// Mitsubishi GX Works2 project: BookEX6_11 Trig   PLC: Q13UDV

// global labels: Global
VAR_GLOBAL
  bVar0 AT M5000 : BOOL;
  abArray0 AT M5010 : ARRAY [0..49] OF BOOL;
  sStr0 AT D5000 : STRING[199];
  sStr1 AT D5100 : STRING[199];
  sStr2 AT D5200 : STRING[199];
  sStr3 AT D5300 : STRING[199];
  sStr4 AT D5400 : STRING[199];
  sStr5 AT D5500 : STRING[199];
  sStr6 AT D5600 : STRING[199];
  sStr7 AT D5700 : STRING[199];
  sStr8 AT D5800 : STRING[199];
  sStr9 AT D5900 : STRING[199];
  iVar0 AT D4500 : INT;
  iVar1 AT D4501 : INT;
  iVar2 AT D4502 : INT;
  iVar3 AT D4503 : INT;
  iVar4 AT D4504 : INT;
  iVar5 AT D4505 : INT;
  iVar6 AT D4506 : INT;
  iVar7 AT D4507 : INT;
  iVar8 AT D4508 : INT;
  iVar9 AT D4509 : INT;
  dVar0 AT D4510 : DINT;
  dVar1 AT D4512 : DINT;
  dVar2 AT D4514 : DINT;
  dVar3 AT D4516 : DINT;
  dVar4 AT D4518 : DINT;
  dVar5 AT D4520 : DINT;
  dVar6 AT D4522 : DINT;
  dVar7 AT D4524 : DINT;
  dVar8 AT D4526 : DINT;
  dVar9 AT D4528 : DINT;
  wVar0 AT D4530 : WORD;
  wVar1 AT D4531 : WORD;
  wVar2 AT D4532 : WORD;
  wVar3 AT D4533 : WORD;
  wVar4 AT D4534 : WORD;
  wVar5 AT D4535 : WORD;
  wVar6 AT D4536 : WORD;
  wVar7 AT D4537 : WORD;
  wVar8 AT D4538 : WORD;
  wVar9 AT D4539 : WORD;
  dwVar0 AT D4540 : DWORD;
  dwVar1 AT D4542 : DWORD;
  dwVar2 AT D4544 : DWORD;
  dwVar3 AT D4546 : DWORD;
  dwVar4 AT D4548 : DWORD;
  dwVar5 AT D4550 : DWORD;
  dwVar6 AT D4552 : DWORD;
  dwVar7 AT D4554 : DWORD;
  dwVar8 AT D4556 : DWORD;
  dwVar9 AT D4558 : DWORD;
  fsVar0 AT D4560 : REAL;
  fsVar1 AT D4562 : REAL;
  fsVar2 AT D4564 : REAL;
  fsVar3 AT D4566 : REAL;
  fsVar4 AT D4568 : REAL;
  fsVar5 AT D4570 : REAL;
  fsVar6 AT D4572 : REAL;
  fsVar7 AT D4574 : REAL;
  fsVar8 AT D4576 : REAL;
  fsVar9 AT D4578 : REAL;
  fdVar0 AT D4580 : LREAL;
  tTime0 AT D4620 : TIME;
  tTime1 AT D4622 : TIME;
  tTime2 AT D4624 : TIME;
  tTime3 AT D4626 : TIME;
  tTime4 AT D4628 : TIME;
  tTime5 AT D4630 : TIME;
  tTime6 AT D4632 : TIME;
  tTime7 AT D4634 : TIME;
  tTime8 AT D4636 : TIME;
  tTime9 AT D4638 : TIME;
  tTime10 AT D4640 : TIME;
  bVar1 AT M5001 : BOOL;
  bVar2 AT M5002 : BOOL;
  bVar3 AT M5003 : BOOL;
  bVar4 AT M5004 : BOOL;
  bVar5 AT M5005 : BOOL;
  bVar6 AT M5006 : BOOL;
  bVar7 AT M5007 : BOOL;
  bVar8 AT M5008 : BOOL;
  bVar9 AT M5009 : BOOL;
  abArray1 AT M5060 : ARRAY [0..49] OF BOOL;
  abArray2 AT M5110 : ARRAY [0..49] OF BOOL;
  abArray3 AT M5160 : ARRAY [0..49] OF BOOL;
  abArray4 AT M5210 : ARRAY [0..49] OF BOOL;
  abArray5 AT M5260 : ARRAY [0..49] OF BOOL;
  abArray6 AT M5310 : ARRAY [0..49] OF BOOL;
  abArray7 AT M5360 : ARRAY [0..49] OF BOOL;
  abArray8 AT M5410 : ARRAY [0..49] OF BOOL;
  abArray9 AT M5460 : ARRAY [0..49] OF BOOL;
  fdVar1 AT D4584 : LREAL;
  fdVar2 AT D4588 : LREAL;
  fdVar3 AT D4592 : LREAL;
  fdVar4 AT D4596 : LREAL;
  fdVar5 AT D4600 : LREAL;
  fdVar6 AT D4604 : LREAL;
  fdVar7 AT D4608 : LREAL;
  fdVar8 AT D4612 : LREAL;
  fdVar9 AT D4616 : LREAL;
  aSendData1 AT D100 : ARRAY [0..9] OF INT;
  aRecvData1 AT D110 : ARRAY [0..9] OF INT;
  aSendData2 AT D120 : ARRAY [0..9] OF INT;
  aRecvData2 AT D130 : ARRAY [0..9] OF INT;
END_VAR
// user libraries (not included): HMI

FUNCTION_BLOCK BiTrig
VAR_INPUT
  b_CK : BOOL;
END_VAR
VAR_OUTPUT
  b_Q : BOOL;
END_VAR
VAR
  oldCK : BOOL;
END_VAR
;
b_Q := b_CK XOR oldCK;
oldCK := b_CK;
END_FUNCTION_BLOCK

FUNCTION_BLOCK FallEdgeTrigger
VAR_INPUT
  b_C : BOOL;
END_VAR
VAR_OUTPUT
  b_F : BOOL;
  b_X : BOOL;
END_VAR
(* structured ladder/FBD written out as ST: instructions are called as NAME(EN, inputs, outputs); _pN, _eN, _tN stand for wires *)
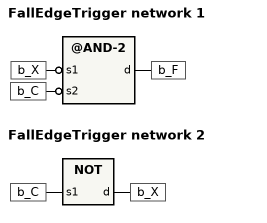
(* network 1 *)
b_F := @AND-2(NOT b_X, NOT b_C);
(* network 2 *)
b_X := NOT(b_C);
END_FUNCTION_BLOCK

FUNCTION_BLOCK real_RTRIG
VAR_INPUT
  fs_D : REAL;
END_VAR
VAR_OUTPUT
  b_Q : BOOL;
END_VAR
VAR_INPUT
  fs_Gap : REAL;
END_VAR
VAR_OUTPUT
  fs_Diff : REAL;
END_VAR
VAR
  fsLast : REAL;
  fsTmp : REAL;
END_VAR
VAR_INPUT
  b_EN : BOOL;
END_VAR
VAR_OUTPUT
  b_ENO : BOOL;
END_VAR
;
b_ENO := b_EN;
IF NOT b_EN THEN
	b_Q := FALSE;
	RETURN;
END_IF;
fsTmp := fs_D - fsLast;
b_Q := ABS(fsTmp) > fs_Gap;
IF b_Q THEN 
	fsLast := fs_D; 
END_IF;
fs_Diff := fs_D - fsLast;
END_FUNCTION_BLOCK

FUNCTION_BLOCK RiseEdgeTrigger
VAR_INPUT
  b_C : BOOL;
END_VAR
VAR_OUTPUT
  b_F : BOOL;
  b_X : BOOL;
END_VAR
(* structured ladder/FBD written out as ST: instructions are called as NAME(EN, inputs, outputs); _pN, _eN, _tN stand for wires *)
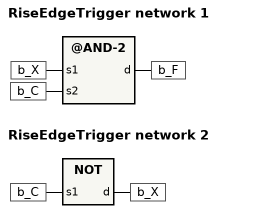
(* network 1 *)
b_F := @AND-2(b_X, b_C);
(* network 2 *)
b_X := NOT(b_C);
END_FUNCTION_BLOCK

FUNCTION_BLOCK sF_TRIG
VAR_INPUT
  b_CK : BOOL;
END_VAR
VAR_OUTPUT
  b_Q : BOOL;
END_VAR
VAR
  oldCK : BOOL;
END_VAR
;
b_Q := NOT b_CK AND NOT oldCK;
oldCK := NOT b_CK;
END_FUNCTION_BLOCK

FUNCTION_BLOCK sR_TRIG
VAR_INPUT
  b_CK : BOOL;
END_VAR
VAR_OUTPUT
  b_Q : BOOL;
END_VAR
VAR
  oldCK : BOOL;
END_VAR
;
b_Q := b_CK AND NOT oldCK;
oldCK := b_CK;
END_FUNCTION_BLOCK

PROGRAM Ex_TRIG
VAR
  F_TRIG_1 : F_TRIG;
  sF_TRIG_1 : sF_TRIG;
  sR_TRIG_1 : sR_TRIG;
  R_TRIG_1 : R_TRIG;
  HMI05_1 : HMI05;
END_VAR
(* structured ladder/FBD written out as ST: instructions are called as NAME(EN, inputs, outputs); _pN, _eN, _tN stand for wires *)
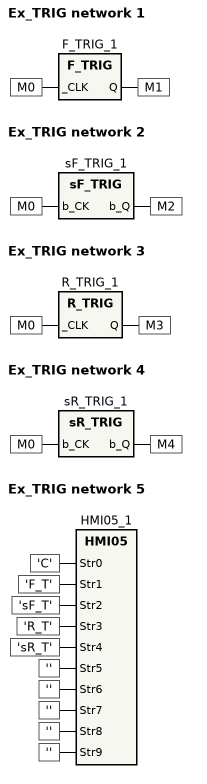
(* network 1 *)
F_TRIG_1(_CLK := M0, Q => M1);
(* network 2 *)
sF_TRIG_1(b_CK := M0, b_Q => M2);
(* network 3 *)
R_TRIG_1(_CLK := M0, Q => M3);
(* network 4 *)
sR_TRIG_1(b_CK := M0, b_Q => M4);
(* network 5 *)
HMI05_1(Str0 := 'C', Str1 := 'F_T', Str2 := 'sF_T', Str3 := 'R_T', Str4 := 'sR_T', Str5 := '', Str6 := '', Str7 := '', Str8 := '', Str9 := '');
END_PROGRAM

PROGRAM ExBiTrig
VAR
  BiTrig_1 : BiTrig;
  HMI05_1 : HMI05;
END_VAR
(* structured ladder/FBD written out as ST: instructions are called as NAME(EN, inputs, outputs); _pN, _eN, _tN stand for wires *)
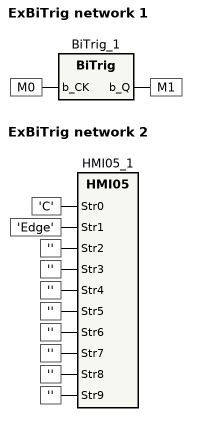
(* network 1 *)
BiTrig_1(b_CK := M0, b_Q => M1);
(* network 2 *)
HMI05_1(Str0 := 'C', Str1 := 'Edge', Str2 := '', Str3 := '', Str4 := '', Str5 := '', Str6 := '', Str7 := '', Str8 := '', Str9 := '');
END_PROGRAM

PROGRAM ExFallEdge
VAR
  FallEdgeTrigger_1 : FallEdgeTrigger;
  FallEdgeTrigger_2 : FallEdgeTrigger;
  F_TRIG_1 : F_TRIG;
  sF_TRIG_1 : sF_TRIG;
  HMI05_1 : HMI05;
END_VAR
(* structured ladder/FBD written out as ST: instructions are called as NAME(EN, inputs, outputs); _pN, _eN, _tN stand for wires *)
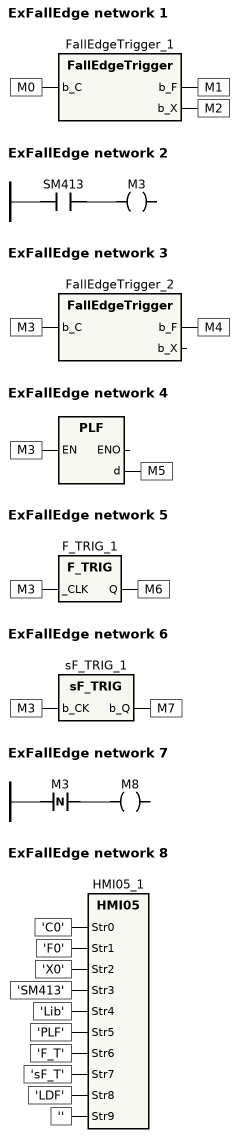
(* network 1 *)
FallEdgeTrigger_1(b_C := M0, b_F => M1, b_X => M2);
(* network 2 *)
M3 := SM413;
(* network 3 *)
FallEdgeTrigger_2(b_C := M3, b_F => M4);
(* network 4 *)
PLF(M3, M5);
(* network 5 *)
F_TRIG_1(_CLK := M3, Q => M6);
(* network 6 *)
sF_TRIG_1(b_CK := M3, b_Q => M7);
(* network 7 *)
M8 := LDF(TRUE, M3);
(* network 8 *)
HMI05_1(Str0 := 'C0', Str1 := 'F0', Str2 := 'X0', Str3 := 'SM413', Str4 := 'Lib', Str5 := 'PLF', Str6 := 'F_T', Str7 := 'sF_T', Str8 := 'LDF', Str9 := '');
END_PROGRAM

PROGRAM ExRealTrig
VAR
  real_RTRIG_1 : real_RTRIG;
  HMI05_1 : HMI05;
END_VAR
(* structured ladder/FBD written out as ST: instructions are called as NAME(EN, inputs, outputs); _pN, _eN, _tN stand for wires *)
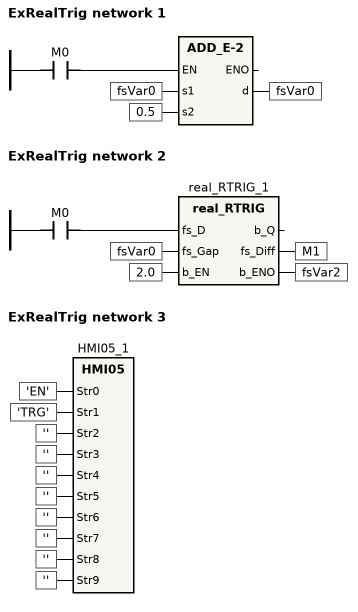
(* network 1 *)
ADD_E(M0, fsVar0, 0.5, fsVar0);
(* network 2 *)
real_RTRIG_1(fs_D := M0, fs_Gap := fsVar0, b_EN := 2.0, fs_Diff => M1, b_ENO => fsVar2);
(* network 3 *)
HMI05_1(Str0 := 'EN', Str1 := 'TRG', Str2 := '', Str3 := '', Str4 := '', Str5 := '', Str6 := '', Str7 := '', Str8 := '', Str9 := '');
END_PROGRAM

PROGRAM ExRiseEdge
VAR
  RiseEdgeTrigger_1 : RiseEdgeTrigger;
  RiseEdgeTrigger_2 : RiseEdgeTrigger;
  FallEdgeTrigger_1 : FallEdgeTrigger;
  FallEdgeTrigger_2 : FallEdgeTrigger;
  R_TRIG_1 : R_TRIG;
  sR_TRIG_1 : sR_TRIG;
  HMI05_1 : HMI05;
END_VAR
(* structured ladder/FBD written out as ST: instructions are called as NAME(EN, inputs, outputs); _pN, _eN, _tN stand for wires *)
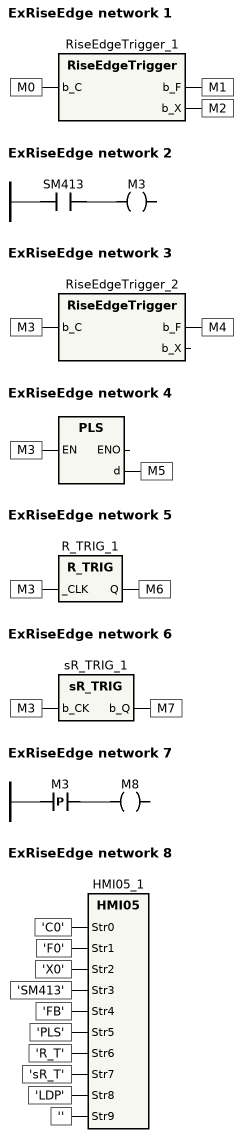
(* network 1 *)
RiseEdgeTrigger_1(b_C := M0, b_F => M1, b_X => M2);
(* network 2 *)
M3 := SM413;
(* network 3 *)
RiseEdgeTrigger_2(b_C := M3, b_F => M4);
(* network 4 *)
PLS(M3, M5);
(* network 5 *)
R_TRIG_1(_CLK := M3, Q => M6);
(* network 6 *)
sR_TRIG_1(b_CK := M3, b_Q => M7);
(* network 7 *)
M8 := LDP(TRUE, M3);
(* network 8 *)
HMI05_1(Str0 := 'C0', Str1 := 'F0', Str2 := 'X0', Str3 := 'SM413', Str4 := 'FB', Str5 := 'PLS', Str6 := 'R_T', Str7 := 'sR_T', Str8 := 'LDP', Str9 := '');
END_PROGRAM

PROGRAM FallEdgeST
VAR
  F_TRIG_1 : F_TRIG;
END_VAR
;
PLF(SM412, M7);
F_TRIG_1(_CLK:=SM412 ,Q:= M8 );
END_PROGRAM

PROGRAM RiseEdgeST
VAR
  R_TRIG_1 : R_TRIG;
END_VAR
;
PLS(SM412, M8);
R_TRIG_1(_CLK:=SM412 ,Q:= M9 );
END_PROGRAM

PROGRAM ExCombo
VAR
  F_TRIG_1 : F_TRIG;
  R_TRIG_1 : R_TRIG;
  HMI05_1 : HMI05;
  F_TRIG_2 : F_TRIG;
  F_TRIG_3 : F_TRIG;
  F_TRIG_4 : F_TRIG;
  R_TRIG_2 : R_TRIG;
  R_TRIG_3 : R_TRIG;
  R_TRIG_4 : R_TRIG;
END_VAR
(* structured ladder/FBD written out as ST: instructions are called as NAME(EN, inputs, outputs); _pN, _eN, _tN stand for wires *)
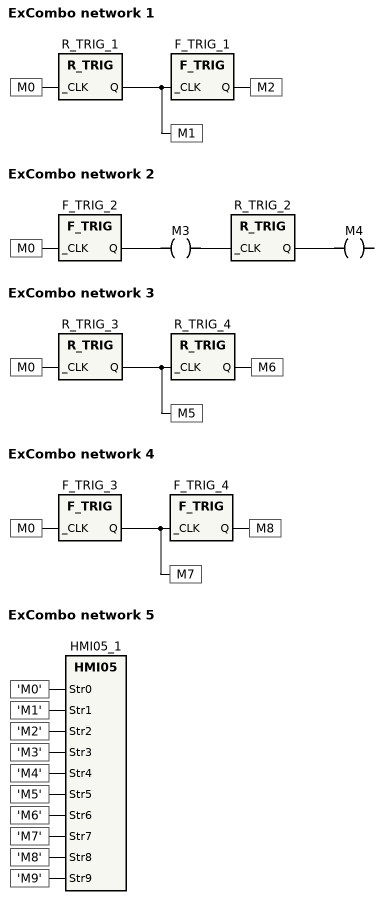
(* network 1 *)
R_TRIG_1(_CLK := M0);
F_TRIG_1(_CLK := R_TRIG_1.Q, Q => M2);
M1 := R_TRIG_1.Q;
(* network 2 *)
F_TRIG_2(_CLK := M0);
M3 := F_TRIG_2.Q;
R_TRIG_2(_CLK := F_TRIG_2.Q);
M4 := R_TRIG_2.Q;
(* network 3 *)
R_TRIG_3(_CLK := M0);
R_TRIG_4(_CLK := R_TRIG_3.Q, Q => M6);
M5 := R_TRIG_3.Q;
(* network 4 *)
F_TRIG_3(_CLK := M0);
F_TRIG_4(_CLK := F_TRIG_3.Q, Q => M8);
M7 := F_TRIG_3.Q;
(* network 5 *)
HMI05_1(Str0 := 'M0', Str1 := 'M1', Str2 := 'M2', Str3 := 'M3', Str4 := 'M4', Str5 := 'M5', Str6 := 'M6', Str7 := 'M7', Str8 := 'M8', Str9 := 'M9');
END_PROGRAM

PROGRAM ExRISE_ST
VAR
  fbButtTrig : R_TRIG;
  bStart : BOOL;
  bCountUp : BOOL;
  iCount : INT;
  fbSenTrig : F_TRIG;
  bSensor : BOOL;
  bNextEn : BOOL;
  bNextMotor : BOOL;
END_VAR
;


fbButtTrig(_CLK := bStart);		

bCountUp := fbButtTrig.Q;		

IF bCountUp THEN				
    iCount := iCount + 1;
END_IF;


fbSenTrig(_CLK := bSensor, Q := bNextEn);		

IF bNextEn THEN			
    bNextMotor := TRUE;
END_IF;
END_PROGRAM
